// TIA Portal V19 export
TYPE "TAx_Speed_Ctrl"
// stored: Access Published
   STRUCT
      SafeStop : Bool;   // 1 = Emergency stop active / Emergency stop (device in safe state)
      Rst : Bool;   // Reset alarms
      RstHW : Bool;   // Reset hardware
      Power : Bool;   // Power axis command
      MovePlus : Bool;
      MoveMinus : Bool;
      ExtControl : Bool;
      Velocity : LReal;
      Acceleration : LReal;
      Deceleration : LReal;
      Jerk : LReal;
   END_STRUCT;
END_TYPE
